FUNCTION UpdateEventTimestampWithSystemTime
VAR_INPUT
	stEvent : REFERENCE TO ST_Event;
END_VAR
VAR
	fbGETSYSTEMTIME : GETSYSTEMTIME;
END_VAR

fbGETSYSTEMTIME()

END_FUNCTION

(* stored: Version 1.1.0.1, ProductVersion 3.1.4024.11
   POU UpdateEventTimestampWithSystemTime: Id {e9b5c6ac-66b4-4e07-ac91-0c1e8bd10fe3}, SpecialFunc None *)
